FUNCTION_BLOCK FB_ConvertUnitsLREALMock EXTENDS FB_FalliblePublicMock IMPLEMENTS I_ConvertUnitsLREAL


METHOD ConvertLREAL
VAR_INPUT
    iQuantity	: I_QuantityLREALPublic;
    sDesiredUnits	: T_MaxString;
END_VAR

iQuantity.Val := iQuantity.Val;
iQuantity.Units := sDesiredUnits;
END_METHOD


METHOD ConvertQuantityLREAL
VAR_INPUT
    QuantityToConvert	: I_QuantityLREAL;
    DesiredUnits	: T_MaxString;
END_VAR
VAR_OUTPUT
    ConvertedQuantity : FB_QuantityLREALPublic(Units := '');
END_VAR

ConvertedQuantity.Val := QuantityToConvert.Val;
ConvertedQuantity.Units := DesiredUnits;
END_METHOD

END_FUNCTION_BLOCK

(* stored: Version 1.1.0.1
   POU FB_ConvertUnitsLREALMock: Id {83003460-d466-485e-a7d1-48cce8fdc0de}, SpecialFunc None
   Method ConvertLREAL: Id {d8395b23-62dd-408a-b46e-942e4ee8a04c}
   Method ConvertQuantityLREAL: Id {7ff13a66-4da9-43c9-a2da-d725026499fd} *)
